PROGRAM prg_AutomatischeDeur
VAR
	bHoofdSchakelaar		AT		%I*			:BOOL;
	bDrukknop				AT		%I*			:BOOL;
	bSensor					AT		%I*			:BOOL;
	
	bDeur					AT		%Q*			:BOOL;
	DeurDicht: TOF;
END_VAR

DeurDicht(IN:= bHoofdSchakelaar AND (bDrukknop OR bSensor), PT:= T#1S, Q=> bDeur);

END_PROGRAM

(* stored: Version 1.1.0.1, ProductVersion 3.1.4024.15
   POU prg_AutomatischeDeur: Id {e8dcdb5a-fded-4c90-a061-70c9e66c14c6}, SpecialFunc None *)
